TYPE EL2809_DEV_CONFIG :
    STRUCT
       
		enableForce	: BOOL;
		forceDigitalOutput_00 : BOOL;
		forceDigitalOutput_01 : BOOL;
		forceDigitalOutput_02 : BOOL;
		forceDigitalOutput_03 : BOOL;
		forceDigitalOutput_04 : BOOL;
		forceDigitalOutput_05 : BOOL;
		forceDigitalOutput_06 : BOOL;
		forceDigitalOutput_07 : BOOL;
		forceDigitalOutput_08 : BOOL;
		forceDigitalOutput_09 : BOOL;
		forceDigitalOutput_10 : BOOL;
		forceDigitalOutput_11 : BOOL;
		forceDigitalOutput_12 : BOOL;
		forceDigitalOutput_13 : BOOL;
		forceDigitalOutput_14 : BOOL;
		forceDigitalOutput_15 : BOOL;
			


    END_STRUCT
END_TYPE

(* stored: Version 1.1.0.1, ProductVersion 3.1.4024.15
   DUT EL2809_DEV_CONFIG: Id {c05184b6-d5bd-488f-9da8-6693691befb6} *)
